(*udt (user defined type) of Beckhoff EL2624 - 4 Point Relay Type Output Terminal:
	Auth: j.vandongen
	October 2019*)


TYPE udt_EP2624_STAT :
STRUCT
	InfoData: udt_ECATSlave_Status;
END_STRUCT
END_TYPE

(* stored: Version 1.1.0.1, ProductVersion 3.1.4024.9
   DUT udt_EP2624_STAT: Id {d629607c-73bc-41f5-8d41-9a436e9acc8d} *)
